(* IEC 61131-3 sources: DataBuffer/src/Ar/DataBuffer, 3 files *)

(* ---- DataBuffer.typ ---- *)
(*
* File: DataBuffer.typ
* Copyright (c) 2023 Loupe
* https://loupe.team
*
* This file is part of DataBuffer, licensed under the MIT License.
*
*)

TYPE
	DATBUF_ERR_enum :
		( (*Status values returned by the DataBuffer functions*)
		DATBUF_ERR_INVALIDINPUT := 50000, (*A required address is 0, or maxLength is 0*)
		DATBUF_ERR_MEMALLOC, (*Memory for the buffer could not be allocated*)
		DATBUF_ERR_NOTINITIALIZED, (*Buffer has not been initialized with datbufInitBuffer*)
		DATBUF_ERR_BUFFERFULL (*Data did not fit in the buffer. The part that fit was appended*)
		);
	datbufBuffer_typ : 	STRUCT  (*Data buffer. Members are maintained by the library*)
		pData : UDINT; (*Address of the data storage. 0 until initialized*)
		currentLength : UDINT; (*Number of bytes of data currently in the buffer [bytes]*)
		maxLength : UDINT; (*Size of the data storage [bytes]*)
	END_STRUCT;
END_TYPE

(* ---- DataBuffer.fun ---- *)
(*
* File: DataBuffer.fun
* Copyright (c) 2023 Loupe
* https://loupe.team
*
* This file is part of DataBuffer, licensed under the MIT License.
*
*)

FUNCTION datbufClearBuffer : UINT (*Reset the buffer length to 0 and zero its data. Returns 0 or a DATBUF_ERR_enum value*) (*$GROUP=User*)
	VAR_INPUT
		pBuffer : UDINT; (*Address of an initialized datbufBuffer_typ*)
	END_VAR
END_FUNCTION

FUNCTION datbufInitBuffer : UINT (*Initialize a data buffer and allocate its memory. Call once, in _INIT. Returns 0 or a DATBUF_ERR_enum value*) (*$GROUP=User*)
	VAR_INPUT
		pBuffer : UDINT; (*Address of the datbufBuffer_typ to initialize*)
		maxLength : UDINT; (*Size of the data storage to allocate [bytes]*)
	END_VAR
END_FUNCTION

FUNCTION datbufAppendToBuffer : UINT (*Append data to a data buffer. Returns 0 or a DATBUF_ERR_enum value*) (*$GROUP=User*)
	VAR_INPUT
		pBuffer : UDINT; (*Address of an initialized datbufBuffer_typ*)
		pData : UDINT; (*Address of the data to append*)
		dataLength : UDINT; (*Length of data to append [bytes]*)
	END_VAR
END_FUNCTION

(* ---- DataBuffer.var ---- *)
(*
* File: DataBuffer.var
* Copyright (c) 2023 Loupe
* https://loupe.team
*
* This file is part of DataBuffer, licensed under the MIT License.
*
*)

VAR CONSTANT

END_VAR
